FUNCTION_BLOCK F_SUM_LAST_N (* Sums up the last N sample values *)
  (* Standard: 61499-2 *)
  (* Version 1.1, 2017-06-15, Marc Jakobi, HTW Berlin *)
  (* Version 1.0, 2016-05-26, AZ, fortiss GmbH *)
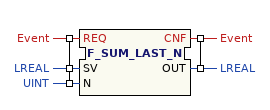
  EVENT_INPUT
    REQ WITH N, SV; (* Normal Execution Request *)
  END_EVENT
  EVENT_OUTPUT
    CNF WITH OUT; (* Execution Confirmation *)
  END_EVENT
  VAR_INPUT
    SV : LREAL; (* New sample value *)
    N : UINT; (* Amount of elements to average over ([1,..,1000]) *)
  END_VAR
  VAR_OUTPUT
    OUT : LREAL; (* Sum of the last N sample values *)
  END_VAR
  VAR
    CACHE : ARRAY [0..9999] OF LREAL; (* Array holding cached data to average over *)
    startIDX : UINT := 0; (* Start index for averaging *)
    endIDX : UINT := 0; (* End index for averaging *)
  END_VAR
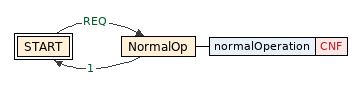
  EC_STATES
    START;
    NormalOp : normalOperation -> CNF; (* Normal execution *)
  END_STATES
  EC_TRANSITIONS
    START TO NormalOp := REQ;
    NormalOp TO START := 1;
  END_TRANSITIONS
  ALGORITHM normalOperation IN ST: (* new algorithm *)
VAR
	j : UINT;
	tmp : UINT;
END_VAR;
// Limit number of values to mean over
IF N > 1000 THEN
	N := 1000;
ELSIF N < 1 THEN
	N := 1;
END_IF;
// Cache current value and increment indexes
CACHE[endIDX] := SV;
// Re-adjust indexes in case N changes
IF endIDX > startIDX THEN // Normal operation
	tmp := endIDX;
ELSE // End of cache passed by endIDX
	tmp := 10000 + endIDX;
END_IF;
IF (tmp - startIDX) > (N - 1) THEN // Increment startIDX to get distance of N values
	WHILE (tmp - startIDX) > (N - 1) DO
		startIDX := startIDX + 1;
			IF startIDX > 9999 THEN // End of CACHE reached
				startIDX := 0;
				tmp := endIDX;
			END_IF;
	END_WHILE;
ELSIF (tmp - startIDX) < (N - 1) THEN // Decrement startIDX to get distance of N values
	WHILE (tmp - startIDX) < (N - 1) DO // Beginning of CACHE reached
		IF startIDX = 0 THEN
			startIDX := 10000;
			tmp := 10000 + endIDX;
		END_IF;
		startIDX := startIDX - 1;
	END_WHILE;
END_IF;
// Sum up last N values
OUT := 0; // Initialize output
IF endIDX >= startIDX THEN // Normal operation
	FOR j := startIDX TO endIDX BY 1 DO
		OUT := OUT + CACHE[j];
	END_FOR;
ELSIF endIDX < startIDX THEN // endIDX moved past end of CACHE
	FOR j := startIDX TO 9999 BY 1 DO // startIDX to end of CACHE
		OUT := OUT + CACHE[j];
	END_FOR;
	FOR j := 0 TO endIDX BY 1 DO // Beginning of CACHE to endIDX
		OUT := OUT + CACHE[j];
	END_FOR;
END_IF;
// Increment endIDX for next request
endIDX := endIDX + 1;
IF endIDX > 9999 THEN // end of CACHE reached
	endIDX := 0;
END_IF;
  END_ALGORITHM
END_FUNCTION_BLOCK
